// TIA Portal V17 export
// export: Created 2024-08-09T12:53:15.4740714Z, ExportSetting WithDefaults, DisplayName Totally Integrated Automation Portal, DisplayVersion V17 Update 7, DisplayName TIA Portal Openness, DisplayVersion V17 Update 7, DisplayName TIA Portal Version Control Interface, DisplayVersion V17, DisplayName STEP 7 Professional, DisplayVersion V17 Update 7, DisplayName STEP 7 Safety, DisplayVersion V17 Update 6, DisplayName WinCC Professional, DisplayVersion V17 Update 7
VAR_GLOBAL   // PLC tag table "Dec_Niveaux_Ensacheuse"
END_VAR
VAR_GLOBAL CONSTANT   // user constants
   NIV_ENS_ATT_DEM_CIR : USInt := 10;
   NIV_ENS_DEM_CIR : USInt := 20;
   NIV_ENS_CIRCUIT_PRET : USInt := 30;
   NIV_ENS_EC : USInt := 40;
   NIV_ENS_VID_CIR : USInt := 50;
   NIV_ENS_ATT_FINLOT : USInt := 60;
   TAC_ENSA1 : SInt := 8;
   TAC_ENSA2 : SInt := 9;
END_VAR
